{attribute 'no_explicit_call' := 'do not call this POU directly'}
FUNCTION_BLOCK T_Logger IMPLEMENTS I_Logger
VAR
    DebugMessage    : T_Message;
    InfoMessage     : T_Message;
    WarningMessage  : T_Message;
    ErrorMessage    : T_Message;
    CriticalMessage : T_Message;

END_VAR

METHOD LogCritical
VAR_INPUT
	Source	: I_TcSourceInfo;
	Message	: Tc2_System.T_MaxString;
END_VAR
CriticalMessage.Send(TcEventSeverity.Critical, Source,Message);
END_METHOD

METHOD LogDebug
VAR_INPUT
	Source	: I_TcSourceInfo;
	Message	: Tc2_System.T_MaxString;
END_VAR
DebugMessage.Send(TcEventSeverity.Verbose, Source,Message);
END_METHOD

METHOD LogError
VAR_INPUT
	Source	: I_TcSourceInfo;
	Message	: Tc2_System.T_MaxString;
END_VAR
ErrorMessage.Send(TcEventSeverity.Error, Source,Message);
END_METHOD

METHOD LogInfo
VAR_INPUT
	Source	: I_TcSourceInfo;
	Message	: Tc2_System.T_MaxString;
END_VAR
InfoMessage.Send(TcEventSeverity.Info, Source,Message);
END_METHOD

METHOD LogWarning
VAR_INPUT
	Source	: I_TcSourceInfo;
	Message	: Tc2_System.T_MaxString;
END_VAR
WarningMessage.Send(TcEventSeverity.Warning, Source,Message);
END_METHOD

END_FUNCTION_BLOCK

(* stored: Version 1.1.0.1, ProductVersion 3.1.4024.15
   POU T_Logger: Id {70ca3160-d298-4ee2-b622-102e6aeec323}, SpecialFunc None
   Method LogCritical: Id {ecb6602c-87f6-49e8-8d1a-1bc5d3deda4c}
   Method LogDebug: Id {ca9e8e2b-0eb7-4666-8779-8521bec7bf46}
   Method LogError: Id {a794fe89-b095-43ad-8664-03e657853ef5}
   Method LogInfo: Id {acc82549-dcc9-4d2d-ab31-37aaa21f9143}
   Method LogWarning: Id {4379dce1-9e59-478f-802e-9722950c9fc6} *)
